PROGRAM Torque_reading
VAR
	MC_TorqueControl_0: MC_TorqueControl;
END_VAR

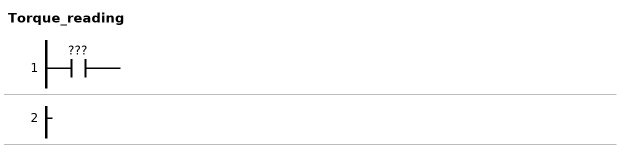
// NETWORK 1

// NETWORK 2

END_PROGRAM

(* stored: Version 1.1.0.1, ProductVersion 3.1.4024.3
   POU Torque_reading: Id {deef73b8-53e6-4cd2-945c-a5a160101c4c}, SpecialFunc None *)
